FUNCTION_BLOCK FB_working
VAR_INPUT
	lightcurtain_mute_left	: BOOL;
	lightcurtain_mute_right	: BOOL;
	pre_tote_status			: ToteStatus;//roller -1 totestatus=ready
	next_tote_status		: ToteStatus;//roller +1 totestatus=empty
END_VAR
VAR_OUTPUT
	status			: MachineStatus := MachineStatus.STOPPED;
	workflow_status	: ToteSubsystemWorkflowStatus := ToteSubsystemWorkflowStatus.UNKNOWN;
	error_status	: OrderToteErrorStatus := OrderToteErrorStatus.UNKNOWN;	
	tote_status		: ToteStatus;
END_VAR
VAR
	current_tote_status	: ToteStatus;
	ton_timeout			: TON;	
	eStates				: E_WorkingStates	:= E_WorkingStates.IDLE;
	eStateTemp			: E_WorkingStates	:= E_WorkingStates.IDLE;
	iStateTemp			: INT;
	sStateTemp			: STRING;
	errorMessage		: STRING;
	xError				: BOOL;
	iMethod_test		: INT;

	xLoading			: BOOL;
	xUnloading			: BOOL;
///////

	valve_lift			: Valve;
	roller_inbound		: Inbound;
	roller_outbound		: Outbound;
	roller_outbound_end	: Outbound;
	sensor_openbag_detection	: ARRAY[0..7] OF BOOL;
	sensor_cover				: ARRAY[0..1] OF BOOL;
	EDM_KA10			: BOOL;
	mcAxis_lift 		: FB_MotionAxis_MC;
	st_mcAxis_lift 		: ST_MotionAxis_MC;
	AxisRef_lift		: AXIS_REF;
	mcAxis_bag 			: FB_MotionAxis_MC;
	st_mcAxis_bag		: ST_MotionAxis_MC;
	AxisRef_bag			: AXIS_REF;	
	event				: ST_EVENT;
	rt_error			: R_TRIG;
	eTransfer			: E_Transfer;
	
	
	bStopped				: BOOL;
END_VAR
VAR CONSTANT
	rPos_lift_up			: REAL	:= 120;
	rPos_lift_down			: REAL	:= 0;
	rPos_bag_opened			: REAL	:= 45;
	rPos_bag_closed			: REAL	:= 0;
	sComponent_name			: STRING := 'fb_working';
END_VAR

M_mapping();

rt_error(CLK:=(roller_inbound.roller.err OR roller_outbound.roller.err OR roller_outbound_end.roller.err OR st_mcAxis_lift.mcReadStatus.Error 
				OR st_mcAxis_bag.mcReadStatus.Error) AND MAIN.eState<>E_SystemManager.RESET_SAFETY);//roller will trig error while power on
IF rt_error.Q THEN
	xError	:= TRUE;
	eStates	:= E_WorkingStates.ERROR;
END_IF

IF NOT(roller_inbound.photo_sensor_mute.Q OR roller_inbound.photo_sensor.Q OR roller_outbound.photo_sensor.Q) THEN
	current_tote_status	:= ToteStatus.EMPTY;
END_IF
IF NOT roller_inbound.photo_sensor_mute.Q AND roller_inbound.photo_sensor.Q AND NOT roller_outbound.photo_sensor.Q THEN
	current_tote_status	:= ToteStatus.READY;
END_IF



IF eStates=E_WorkingStates.IDLE THEN
	bStopped	:= TRUE;
ELSE
	bStopped	:= FALSE;
END_IF
CASE iMethod_test OF
	0:
	;
	1:		
		IF 	M_load() THEN
			iMethod_test	:= 0;
		END_IF
	2:
		IF 	M_bag_open() THEN
			iMethod_test	:= 0;
		END_IF
	3:
		IF 	M_unload() THEN
			iMethod_test	:= 0;
		END_IF
		
END_CASE

METHOD M_agingTest : BOOL
VAR_INPUT
	
END_VAR
M_AgingTest	:= FALSE;
//////////////////////////////////////////////////////////timeout//////////////////////////////////////////
iStateTemp	:= eStateTemp;
ton_timeout();
IF eStates<>E_WorkingStates.IDLE AND eStates<>E_WorkingStates.ERROR THEN
	IF eStateTemp=eStates THEN
		ton_timeout.IN	:=TRUE;
	ELSE
		ton_timeout.IN	:=FALSE;
		eStateTemp	:= eStates;
	END_IF
ELSE
	ton_timeout.IN	:=FALSE;
END_IF
IF ton_timeout.Q THEN	
	ton_timeout.IN	:=FALSE;
	CASE eStates OF
		E_WorkingStates.AGING_STATE_0:		
			errorMessage	:= CONCAT('wait loading timeout.->fb_loading ',INT_TO_STRING(iStateTemp));
		E_WorkingStates.AGING_STATE_1:		
			errorMessage	:= CONCAT('wait unloading timeout.->fb_loading ',INT_TO_STRING(iStateTemp));
	END_CASE
	IF eStates<>E_WorkingStates.WAIT AND eStates<>E_WorkingStates.WAIT_1 THEN
		//eStates	:= E_WorkingStates.ERROR;
		;
	END_IF
END_IF
CASE eStates OF
	E_WorkingStates.IDLE:
		eStates	:= E_WorkingStates.AGING_STATE_0;
	E_WorkingStates.AGING_STATE_0:
		ton_timeout.PT	:= T#2S;
		st_mcAxis_bag.mcMoveAbsolute.Execute	:= TRUE;						
		st_mcAxis_bag.rActualPosSet	:= rPos_bag_closed;
		st_mcAxis_bag.rVelocitySet	:= 100;
		st_mcAxis_lift.mcMoveAbsolute.Execute	:= TRUE;	
		st_mcAxis_lift.rActualPosSet	:= rPos_lift_up;
		st_mcAxis_lift.rVelocitySet	:= 100;	
		roller_inbound.roller.forward			:= TRUE;
		roller_inbound.roller.backward			:= FALSE;
		roller_outbound.roller.forward			:= TRUE;
		roller_outbound_end.roller.forward		:= TRUE;
		roller_outbound_end.roller.backward		:= FALSE;			
		IF st_mcAxis_bag.mcMoveAbsolute.Done AND st_mcAxis_lift.mcMoveAbsolute.Done AND ton_timeout.Q THEN
			eStates	:= E_WorkingStates.WAIT;
		END_IF			
	E_WorkingStates.WAIT:
		roller_inbound.roller.forward			:= FALSE;
		roller_inbound.roller.backward			:= FALSE;
		roller_outbound.roller.forward			:= FALSE;
		roller_outbound.roller.backward			:= FALSE;
		roller_outbound_end.roller.forward		:= FALSE;
		roller_outbound_end.roller.backward		:= FALSE;	
		st_mcAxis_bag.mcMoveAbsolute.Execute	:= FALSE;
		st_mcAxis_lift.mcMoveAbsolute.Execute	:= FALSE;		
		ton_timeout.PT	:= T#1S;
		IF ton_timeout.Q THEN
			eStates	:= E_WorkingStates.AGING_STATE_1;
		END_IF
	E_WorkingStates.AGING_STATE_1:
		ton_timeout.PT	:= T#2S;
		st_mcAxis_bag.mcMoveAbsolute.Execute	:= TRUE;						
		st_mcAxis_bag.rActualPosSet	:= rPos_bag_opened;
		st_mcAxis_bag.rVelocitySet	:= 100;
		st_mcAxis_lift.mcMoveAbsolute.Execute	:= TRUE;
		st_mcAxis_lift.rActualPosSet	:= rPos_lift_down;
		st_mcAxis_lift.rVelocitySet	:= 100;	
		roller_inbound.roller.forward			:= TRUE;
		roller_inbound.roller.backward			:= TRUE;
		roller_outbound.roller.backward			:= TRUE;
		roller_outbound_end.roller.forward		:= TRUE;
		roller_outbound_end.roller.backward		:= TRUE;			
		IF st_mcAxis_bag.mcMoveAbsolute.Done AND st_mcAxis_lift.mcMoveAbsolute.Done AND ton_timeout.Q THEN
			eStates	:= E_WorkingStates.WAIT_1;
		END_IF	
	E_WorkingStates.WAIT_1:
		ton_timeout.PT	:= T#1S;
		roller_inbound.roller.forward			:= FALSE;
		roller_inbound.roller.backward			:= FALSE;
		roller_outbound.roller.forward			:= FALSE;
		roller_outbound.roller.backward			:= FALSE;
		roller_outbound_end.roller.forward		:= FALSE;
		roller_outbound_end.roller.backward		:= FALSE;	
		st_mcAxis_bag.mcMoveAbsolute.Execute	:= FALSE;
		st_mcAxis_lift.mcMoveAbsolute.Execute	:= FALSE;		
		IF ton_timeout.Q THEN
			eStates	:= E_WorkingStates.IDLE;
		END_IF		
	E_WorkingStates.DONE:
		;
	E_WorkingStates.ERROR:
		;
	
END_CASE
END_METHOD

METHOD M_bag_close : BOOL
VAR_INPUT
END_VAR
END_METHOD

METHOD M_bag_open : BOOL
VAR_INPUT
END_VAR
M_bag_open	:= FALSE;
ADSLOGSTR(msgCtrlMask:= ADSLOG_MSGTYPE_LOG,msgFmtStr:='bag open',strArg:='MSG ARG');
M_bag_open	:= TRUE;
END_METHOD

METHOD M_checkCondition : BOOL
VAR_INPUT
	condition	: E_Condition;
END_VAR
M_checkCondition	:= FALSE;
CASE condition OF
	E_Condition.NO_TOTE:
	 	IF NOT roller_inbound.photo_sensor.Q THEN
			M_checkCondition	:= TRUE;
		END_IF
	E_Condition.TOTE_IN:
	 	IF roller_inbound.photo_sensor.Q THEN
			M_checkCondition	:= TRUE;
		END_IF		
	E_Condition.READY_LOADING_TOTE:
		IF pre_tote_status=ToteStatus.READY THEN
			M_checkCondition	:= TRUE;
		END_IF
	E_Condition.TOTE_READY:
		IF ABS(st_mcAxis_lift.mcReadActualPosition.Position-rPos_lift_down)<1 AND ABS(st_mcAxis_bag.mcReadActualPosition.Position-rPos_bag_opened)<1 
			AND roller_inbound.photo_sensor.Q AND NOT roller_inbound.photo_sensor_mute.Q AND NOT roller_outbound.photo_sensor.Q AND valve_lift.retracted THEN
			tote_status	:= ToteStatus.READY;
		ELSE
			IF tote_status = ToteStatus.READY THEN
				tote_status	:= ToteStatus.LOADED;
			END_IF
		END_IF
		IF ABS(st_mcAxis_lift.mcReadActualPosition.Position-rPos_lift_up)<1 AND ABS(st_mcAxis_bag.mcReadActualPosition.Position-rPos_bag_closed)<1 
			AND NOT roller_inbound.photo_sensor.Q AND NOT roller_inbound.photo_sensor_mute.Q AND NOT roller_outbound.photo_sensor.Q AND valve_lift.retracted THEN
			tote_status	:= ToteStatus.EMPTY;	
		END_IF	
		M_checkCondition	:= TRUE;
END_CASE
END_METHOD

METHOD M_init : BOOL
VAR_INPUT
END_VAR
M_init	:= FALSE;
event.sMethod	:= 'init';
xError	:= FALSE;
st_mcAxis_bag.mcStop.Execute	:= FALSE;
st_mcAxis_bag.mcReset.Execute	:= TRUE;
st_mcAxis_lift.mcStop.Execute	:= FALSE;
st_mcAxis_lift.mcReset.Execute	:= TRUE;
error_status	:= OrderToteErrorStatus.NO_ERROR;

eStates	:= E_WorkingStates.IDLE;
M_init	:= TRUE;
END_METHOD

METHOD M_load : BOOL
VAR_INPUT
END_VAR
VAR_OUTPUT 

END_VAR
M_load := FALSE;
event.sMethod	:= 'load';
//////////////////////////////////////////////////////////timeout//////////////////////////////////////////
iStateTemp	:= eStateTemp;
sStateTemp	:= INT_TO_STRING(iStateTemp);
ton_timeout();
IF eStates<>E_WorkingStates.IDLE AND eStates<>E_WorkingStates.ERROR THEN
	IF eStateTemp=eStates THEN
		ton_timeout.IN	:=TRUE;
	ELSE
		ton_timeout.IN	:=FALSE;
		IF GVL.bAck_stop THEN
			roller_inbound.roller.forward	:= FALSE;
			RETURN;			
		END_IF
		eStateTemp	:= eStates;	
	END_IF
ELSE
	ton_timeout.IN	:=FALSE;
END_IF
IF ton_timeout.Q THEN	
	ton_timeout.IN	:=FALSE;
	CASE eStates OF		
		E_WorkingStates.BAG_OPEN_UP:	
			event.sEventType	:= 'error';
			event.sEvent_MSG	:= CONCAT('BAG_OPEN_UP ','timeout');
			event.sStepID		:= sStateTemp;
		E_WorkingStates.BAG_CLOSE:	
			event.sEventType	:= 'error';
			event.sEvent_MSG	:= CONCAT('BAG_CLOSE ','timeout');
			event.sStepID		:= sStateTemp;					
		E_WorkingStates.TOTE_LIFT_DOWN:			
			event.sEventType	:= 'error';
			event.sEvent_MSG	:= CONCAT('TOTE_LIFT_DOWN ','timeout');
			event.sStepID		:= sStateTemp;
		E_WorkingStates.WAIT_NEW_TOTE://wait empty and trig signal
			;
		E_WorkingStates.TOTE_LOAD:	
			event.sEventType	:= 'error';
			event.sEvent_MSG	:= CONCAT('TOTE_LOAD ','timeout');
			event.sStepID		:= sStateTemp;
		E_WorkingStates.WAIT:
			;
		E_WorkingStates.BAG_OPEN_DOWN:
			event.sEventType	:= 'error';
			event.sEvent_MSG	:= CONCAT('BAG_OPEN_DOWN ','timeout');
			event.sStepID		:= sStateTemp;			
		E_WorkingStates.BAG_OPEN:			
			event.sEventType	:= 'error';
			event.sEvent_MSG	:= CONCAT('BAG_OPEN ','timeout');
			event.sStepID		:= sStateTemp;
		ELSE
			event.sEventType	:= 'error';
			event.sEvent_MSG	:= CONCAT('unknow estate ','timeout');
			event.sStepID		:= sStateTemp;			
	END_CASE
	IF eStates<>E_WorkingStates.WAIT_NEW_TOTE AND eStates<>E_WorkingStates.WAIT THEN
		eStates	:= E_WorkingStates.ERROR;
		error_status	:= OrderToteErrorStatus.MECHANICAL_ERROR;
		Event_add(event);
	END_IF
	
END_IF

CASE eStates OF 
		E_WorkingStates.IDLE:
			ton_timeout.PT	:= T#10S;
			xLoading	:= FALSE;
			xUnloading	:= FALSE;
			st_mcAxis_bag.mcPower.Enable	:= TRUE;
			st_mcAxis_lift.mcPower.Enable	:= TRUE;
			IF st_mcAxis_bag.mcReadStatus.StandStill AND st_mcAxis_lift.mcReadStatus.StandStill THEN
				eStates	:= E_WorkingStates.INIT;
			END_IF			
		E_WorkingStates.INIT:
			xLoading	:= TRUE;		
			st_mcAxis_bag.mcMoveAbsolute.Execute	:= FALSE;
			st_mcAxis_lift.mcMoveAbsolute.Execute	:= FALSE;
			eStates	:= E_WorkingStates.BAG_OPEN_UP;
		E_WorkingStates.BAG_OPEN_UP:	
			st_mcAxis_lift.mcMoveAbsolute.Execute	:= TRUE;		
			st_mcAxis_lift.rActualPosSet	:= rPos_lift_up;
			st_mcAxis_lift.rVelocitySet	:= 250;
			IF st_mcAxis_lift.mcMoveAbsolute.Done THEN
				st_mcAxis_lift.mcMoveAbsolute.Execute	:= FALSE;
				eStates	:= E_WorkingStates.BAG_CLOSE;
			END_IF	
		E_WorkingStates.BAG_CLOSE:	
			st_mcAxis_bag.mcMoveAbsolute.Execute	:= TRUE;		
			st_mcAxis_bag.rActualPosSet	:= rPos_bag_closed;
			st_mcAxis_bag.rVelocitySet	:= 250;
			IF st_mcAxis_bag.mcMoveAbsolute.Done THEN
				st_mcAxis_bag.mcMoveAbsolute.Execute	:= FALSE;
				eStates	:= E_WorkingStates.TOTE_LIFT_DOWN;
			END_IF					
		E_WorkingStates.TOTE_LIFT_DOWN:			
			valve_lift.extend	:= FALSE;
			valve_lift.retract	:= TRUE;
			IF NOT valve_lift.extended AND valve_lift.retracted THEN
				eStates	:= E_WorkingStates.WAIT_NEW_TOTE;
			END_IF	
		E_WorkingStates.WAIT_NEW_TOTE://wait empty and trig signal
			workflow_status	:= ToteSubsystemWorkflowStatus.WAITING_FOR_NEW_TOTE;
			IF NOT(roller_inbound.photo_sensor_mute.Q OR roller_inbound.photo_sensor.Q OR roller_outbound.photo_sensor.Q) THEN
				tote_status	:= ToteStatus.EMPTY;
			END_IF
			IF M_waitCondition(condition:=E_Condition.READY_LOADING_TOTE) THEN
				eStates	:= E_WorkingStates.TOTE_LOAD;
			END_IF
		E_WorkingStates.TOTE_LOAD:	
			workflow_status	:= ToteSubsystemWorkflowStatus.INBOUNDING;
			ton_timeout.PT	:= T#10S;	
			roller_inbound.roller.forward	:= TRUE;
			IF roller_inbound.photo_sensor.Q THEN	
				eStates	:= E_WorkingStates.WAIT;
			END_IF
		E_WorkingStates.WAIT:
			ton_timeout.PT	:= T#300MS;
			roller_inbound.roller.forward	:= TRUE;
			IF ton_timeout.Q THEN
				tote_status	:= ToteStatus.LOADED;
				roller_inbound.roller.forward	:= FALSE;
				eStates	:= E_WorkingStates.BAG_OPEN_DOWN;
			END_IF
		E_WorkingStates.BAG_OPEN_DOWN:
			ton_timeout.PT	:= T#10S;
			workflow_status	:= ToteSubsystemWorkflowStatus.BAG_OPENING;
			st_mcAxis_lift.mcMoveAbsolute.Execute	:= TRUE;		
			st_mcAxis_lift.rActualPosSet	:= rPos_lift_down;
			st_mcAxis_lift.rVelocitySet	:= 250;
			IF st_mcAxis_lift.mcMoveAbsolute.Done THEN
				st_mcAxis_bag.mcMoveAbsolute.Execute	:= FALSE;
				eStates	:= E_WorkingStates.BAG_OPEN;
			END_IF			
		E_WorkingStates.BAG_OPEN:			
			st_mcAxis_bag.mcMoveAbsolute.Execute	:= TRUE;		
			st_mcAxis_bag.rActualPosSet	:= rPos_bag_opened;
			st_mcAxis_bag.rVelocitySet	:= 250;
			IF st_mcAxis_bag.mcMoveAbsolute.Done THEN
				st_mcAxis_bag.mcMoveAbsolute.Execute	:= FALSE;
				eStates	:= E_WorkingStates.DONE;
			END_IF
		E_WorkingStates.DONE:
			tote_status	:= ToteStatus.READY;
			workflow_status	:= ToteSubsystemWorkflowStatus.IDLE;	
			M_load	:= TRUE;
			xLoading	:= FALSE;
			eStates	:= E_WorkingStates.IDLE;
		E_WorkingStates.ERROR:
			xError	:=	TRUE;
			workflow_status	:= ToteSubsystemWorkflowStatus.IDLE;
			roller_inbound.roller.forward		:= FALSE;	
			st_mcAxis_bag.mcMoveAbsolute.Execute	:= FALSE;
			st_mcAxis_lift.mcMoveAbsolute.Execute	:= FALSE;			
			M_load 		:= TRUE;
		
END_CASE
END_METHOD

METHOD M_mapping : BOOL
VAR_INPUT
END_VAR
event.sTime	:= MAIN.Temp_str;
event.sComponent_name	:= sComponent_name;
/////////////////////////////////////digital input////////////////////////////////////////
valve_lift.extended					:= G_IO.arDI[5].Ch[0] OR G_IO.arDI[5].Ch[2];
valve_lift.retracted				:= G_IO.arDI[5].Ch[1] OR G_IO.arDI[5].Ch[3];
roller_inbound.photo_sensor_mute(D:= G_IO.arDI[5].Ch[4],on_ms:=10,off_ms:=100);
roller_inbound.roller.err			:= G_IO.arDI[5].Ch[5];
roller_inbound.photo_sensor(D:= G_IO.arDI[5].Ch[6],on_ms:=100,off_ms:=100);
roller_outbound.roller.err			:= G_IO.arDI[5].Ch[7];
roller_outbound.photo_sensor(D:= G_IO.arDI[5].Ch[8],on_ms:=100,off_ms:=500);		
sensor_openbag_detection[0]			:= G_IO.arDI[5].Ch[9];
sensor_openbag_detection[1]			:= G_IO.arDI[5].Ch[10];
sensor_openbag_detection[2]			:= G_IO.arDI[5].Ch[11];
sensor_openbag_detection[3]			:= G_IO.arDI[5].Ch[12];
sensor_openbag_detection[4]			:= G_IO.arDI[5].Ch[13];
sensor_openbag_detection[5]			:= G_IO.arDI[5].Ch[14];
sensor_openbag_detection[6]			:= G_IO.arDI[5].Ch[15];
sensor_openbag_detection[7]			:= G_IO.arDI[6].Ch[0];
sensor_cover[0]						:= G_IO.arDI[6].Ch[1];
sensor_cover[1]						:= G_IO.arDI[6].Ch[2];
EDM_KA10							:= G_IO.arDI[6].Ch[3];
roller_outbound_end.roller.err		:= G_IO.arDI[6].Ch[4];


/////////////////////////////////////digital output////////////////////////////////////////
G_IO.arDO[5].Ch[0]	:= valve_lift.extend;
G_IO.arDO[5].Ch[1]	:= valve_lift.retract;
G_IO.arDO[5].Ch[2]	:= roller_inbound.roller.forward;
G_IO.arDO[5].Ch[3]	:= roller_inbound.roller.backward;
G_IO.arDO[5].Ch[4]	:= roller_outbound.roller.forward;
G_IO.arDO[5].Ch[5]	:= roller_outbound.roller.backward;
G_IO.arDO[5].Ch[6]	:= roller_outbound_end.roller.forward;
G_IO.arDO[5].Ch[7]	:= roller_outbound_end.roller.backward;
G_IO.arDO[5].Ch[8]	:= lightcurtain_mute_left;
G_IO.arDO[5].Ch[9]	:= lightcurtain_mute_right;



/////////////////////////////////////axis config////////////////////////////////////////
mcAxis_lift
(
	ZSN		:=  TRUE OR st_mcAxis_lift.xHoming, //TODO link to digital input
	ZSP		:=  TRUE OR st_mcAxis_lift.xHoming, //TODO link to digital input
	IN_OUT	:= st_mcAxis_lift	, 
	AXIS	:= AxisRef_lift	, 
);
st_mcAxis_lift.bPosSensorShow	:= TRUE;
st_mcAxis_lift.bNegSensorShow	:= TRUE;
st_mcAxis_lift.rMaxAcceleration	:= 50000;
st_mcAxis_lift.rMaxDeceleration	:= 50000;
st_mcAxis_lift.rMaxJerk			:= 500000;
st_mcAxis_lift.rAcceleration	:= 2500;
st_mcAxis_lift.rDeceleration	:= 2500;
st_mcAxis_lift.rJerk			:= 12500;
st_mcAxis_lift.rMaxVelocity		:= 100;
st_mcAxis_lift.rMaxDistance		:= 50;
st_mcAxis_lift.bPosSen	:= TRUE ;//TODO link to digital input
st_mcAxis_lift.bNegSen	:= TRUE ;//TODO link to digital input
st_mcAxis_lift.mcHome.bCalibrationCam	:= TRUE;//TODO link to digital input origin
st_mcAxis_lift.bPositionSensor	:= TRUE;//TODO link to digital input origin
st_mcAxis_lift.bdirFW	:= TRUE;
st_mcAxis_lift.sNetID := '192.168.11.159.5.1';
st_mcAxis_lift.nSlaveAddr	:= 1026;


mcAxis_bag
(
	ZSN		:=  TRUE OR st_mcAxis_bag.xHoming, //TODO link to digital input
	ZSP		:=  TRUE OR st_mcAxis_bag.xHoming, //TODO link to digital input
	IN_OUT	:= st_mcAxis_bag	, 
	AXIS	:= AxisRef_bag	, 
);
st_mcAxis_bag.bPosSensorShow	:= TRUE;
st_mcAxis_bag.bNegSensorShow	:= TRUE;
st_mcAxis_bag.rMaxAcceleration	:= 50000;
st_mcAxis_bag.rMaxDeceleration	:= 50000;
st_mcAxis_bag.rMaxJerk			:= 500000;
st_mcAxis_bag.rAcceleration	:= 2500;
st_mcAxis_bag.rDeceleration	:= 2500;
st_mcAxis_bag.rJerk			:= 12500;
st_mcAxis_bag.rMaxVelocity		:= 100;
st_mcAxis_bag.rMaxDistance		:= 50;
st_mcAxis_bag.bPosSen	:= TRUE ;//TODO link to digital input
st_mcAxis_bag.bNegSen	:= TRUE ;//TODO link to digital input
st_mcAxis_bag.mcHome.bCalibrationCam	:= TRUE;//TODO link to digital input origin
st_mcAxis_bag.bPositionSensor	:= TRUE;//TODO link to digital input origin
st_mcAxis_bag.bdirFW	:= TRUE;
st_mcAxis_bag.sNetID := '192.168.11.159.5.1';
st_mcAxis_bag.nSlaveAddr	:= 1027;

IF MAIN.firstCycle THEN
	st_mcAxis_bag.mcPower.Enable	:= TRUE;
	st_mcAxis_lift.mcPower.Enable	:= TRUE;	
END_IF
END_METHOD

METHOD M_reset : BOOL
VAR_INPUT
END_VAR
M_reset	:= FALSE;
ton_timeout.IN	:= FALSE;
event.sMethod	:= 'reset';
error_status	:= OrderToteErrorStatus.NO_ERROR;
IF xError THEN
	st_mcAxis_bag.mcStop.Execute	:= FALSE;
	st_mcAxis_bag.mcReset.Execute	:= TRUE;
	st_mcAxis_lift.mcStop.Execute	:= FALSE;
	st_mcAxis_lift.mcReset.Execute	:= TRUE;
	IF eStates<>E_WorkingStates.IDLE THEN
		eStates	:= eStateTemp;//continue
	END_IF
		
	xError	:= FALSE;
ELSE
	;
END_IF

//todo:check if reset successful
M_reset	:= TRUE;
END_METHOD

METHOD M_run : BOOL
VAR_INPUT
END_VAR
//
IF M_checkCondition(condition:= E_Condition.NO_TOTE) THEN
	;
END_IF
//check no tote of working
//wait new tote of loading
//tote load
END_METHOD

METHOD M_runStart : BOOL
VAR_INPUT
END_VAR
M_runStart	:= FALSE;
st_mcAxis_bag.mcPower.Enable	:= TRUE;
st_mcAxis_lift.mcPower.Enable	:= TRUE;

current_tote_status	:= ToteStatus.UNKNOWN;
M_checkCondition(condition:=E_Condition.TOTE_READY);


IF st_mcAxis_bag.mcReadStatus.StandStill AND st_mcAxis_lift.mcReadStatus.StandStill THEN
	M_runStart	:= TRUE;
END_IF
M_runStart	:= TRUE;
END_METHOD

METHOD M_safetyEvent : BOOL
VAR_INPUT
END_VAR
M_safetyEvent	:= FALSE;

roller_inbound.roller.forward			:= FALSE;
roller_inbound.roller.backward			:= FALSE;
roller_outbound.roller.forward			:= FALSE;
roller_outbound.roller.backward			:= FALSE;
roller_outbound_end.roller.forward		:= FALSE;	
roller_outbound_end.roller.backward		:= FALSE;	
st_mcAxis_bag.mcMoveAbsolute.Execute	:= FALSE;
st_mcAxis_lift.mcMoveAbsolute.Execute	:= FALSE;	
st_mcAxis_bag.mcStop.Execute	:= TRUE;
st_mcAxis_lift.mcStop.Execute	:= TRUE;

M_safetyEvent	:= TRUE;
END_METHOD

METHOD M_toteLoad : BOOL
VAR_INPUT
END_VAR
M_toteLoad	:= FALSE;
IF roller_inbound.photo_sensor.Q THEN
	roller_inbound.roller.forward	:= FALSE;
	ADSLOGSTR(msgCtrlMask:= ADSLOG_MSGTYPE_LOG,msgFmtStr:='tote load finish',strArg:='MSG ARG');
ELSE
	roller_inbound.roller.forward	:= TRUE;
	ADSLOGSTR(msgCtrlMask:= ADSLOG_MSGTYPE_LOG,msgFmtStr:='tote load start',strArg:='MSG ARG');
	M_toteLoad	:= TRUE;
END_IF
END_METHOD

METHOD M_toteUnload : BOOL
VAR_INPUT
END_VAR
M_toteUnload	:= FALSE;

CASE eStates OF 
		E_WorkingStates.TOTE_LIFT_UP:
			valve_lift.extend	:= TRUE;
			valve_lift.retract	:= FALSE;
			IF valve_lift.extended AND NOT valve_lift.retracted THEN
				eStates	:= E_WorkingStates.TOTE_UNLOAD;
			END_IF
		E_WorkingStates.TOTE_OUT:
			IF roller_outbound.photo_sensor.Q THEN
				roller_outbound.roller.forward	:= FALSE;
				M_toteUnload	:= TRUE;
			ELSE
				roller_outbound.roller.forward	:= TRUE;
			END_IF	
		E_WorkingStates.TOTE_LIFT_DOWN:	
			valve_lift.extend	:= FALSE;
			valve_lift.retract	:= TRUE;
			IF NOT valve_lift.extended AND valve_lift.retracted THEN
				M_toteUnload	:= TRUE;
			END_IF	
END_CASE
END_METHOD

METHOD M_unload : BOOL
VAR_INPUT
END_VAR
VAR_OUTPUT 

END_VAR
//initialize
//bag_open lift up & bag_open_home
//tote lift up
//outbound
//tote lift down
//done
M_unload := FALSE;
event.sMethod	:= 'unload';
//////////////////////////////////////////////////////////timeout//////////////////////////////////////////
iStateTemp	:= eStateTemp;
sStateTemp	:= INT_TO_STRING(iStateTemp);
ton_timeout();
IF eStates<>E_WorkingStates.IDLE AND eStates<>E_WorkingStates.ERROR  THEN
	IF eStateTemp=eStates THEN
		ton_timeout.IN	:=TRUE;
	ELSE
		ton_timeout.IN	:=FALSE;
		IF GVL.bAck_stop THEN
			roller_outbound.roller.forward	:= FALSE;
			roller_outbound_end.roller.forward	:= FALSE;
			RETURN;		
		END_IF
		eStateTemp	:= eStates;
	END_IF
ELSE
	ton_timeout.IN	:=FALSE;
END_IF
IF ton_timeout.Q THEN	
	ton_timeout.IN	:=FALSE;
	CASE eStates OF
	
		E_WorkingStates.WAIT_UNLOADING://wait signal from logtech and app to unload the tote
			;
		E_WorkingStates.BAG_OPEN_UP:	
			event.sEventType	:= 'error';
			event.sEvent_MSG	:= CONCAT('BAG_OPEN_UP ','timeout');
			event.sStepID		:= sStateTemp;
		E_WorkingStates.BAG_CLOSE:	
			event.sEventType	:= 'error';
			event.sEvent_MSG	:= CONCAT('BAG_CLOSE or TOTE_LIFT_UP ','timeout');
			event.sStepID		:= sStateTemp;						
		E_WorkingStates.TOTE_LIFT_UP:
			event.sEventType	:= 'error';
			event.sEvent_MSG	:= CONCAT('TOTE_LIFT_UP ','timeout');
			event.sStepID		:= sStateTemp;
		E_WorkingStates.TOTE_UNLOAD:
			event.sEventType	:= 'error';
			event.sEvent_MSG	:= CONCAT('TOTE_UNLOAD ','timeout');
			event.sStepID		:= sStateTemp;

		E_WorkingStates.WAIT_SENSOR_OFF:	
			event.sEventType	:= 'error';
			event.sEvent_MSG	:= CONCAT('WAIT_SENSOR_OFF ','timeout');
			event.sStepID		:= sStateTemp;	
		E_WorkingStates.TOTE_LIFT_DOWN:
			event.sEventType	:= 'error';
			event.sEvent_MSG	:= CONCAT('TOTE_LIFT_DOWN ','timeout');
			event.sStepID		:= sStateTemp;
		ELSE
			event.sEventType	:= 'error';
			event.sEvent_MSG	:= CONCAT('unknow estate ','timeout');
			event.sStepID		:= sStateTemp;			
	END_CASE
	IF eStates<>E_WorkingStates.IDLE AND eStates<>E_WorkingStates.WAIT_UNLOADING THEN
		eStates	:= E_WorkingStates.ERROR;
		error_status	:= OrderToteErrorStatus.MECHANICAL_ERROR;
		Event_add(event);
	END_IF
	
END_IF

CASE eStates OF 
		E_WorkingStates.IDLE:
			ton_timeout.PT	:= T#10S;
			xLoading	:= FALSE;
			xUnloading	:= FALSE;
			eStates	:= E_WorkingStates.INIT;
		E_WorkingStates.INIT:	
			xUnloading	:= TRUE;
			st_mcAxis_bag.mcMoveAbsolute.Execute	:= FALSE;
			st_mcAxis_lift.mcMoveAbsolute.Execute	:= FALSE;
			eStates	:= E_WorkingStates.WAIT_UNLOADING;
		E_WorkingStates.WAIT_UNLOADING://wait signal from logtech and app to unload the tote
			workflow_status	:= ToteSubsystemWorkflowStatus.WAITING_FOR_UNLOADING;
			tote_status	:= ToteStatus.READY;
			eStates	:= E_WorkingStates.BAG_OPEN_UP;	
		E_WorkingStates.BAG_OPEN_UP:	
			workflow_status	:= ToteSubsystemWorkflowStatus.OUTBOUNDING;	
			tote_status	:= ToteStatus.LOADED;		
			st_mcAxis_lift.mcMoveAbsolute.Execute	:= TRUE;		
			st_mcAxis_lift.rActualPosSet	:= rPos_lift_up;
			st_mcAxis_lift.rVelocitySet	:= 250;
			IF st_mcAxis_lift.mcMoveAbsolute.Done THEN
				eStates	:= E_WorkingStates.BAG_CLOSE;
			END_IF		
		E_WorkingStates.BAG_CLOSE:	
			st_mcAxis_bag.mcMoveAbsolute.Execute	:= TRUE;		
			st_mcAxis_bag.rActualPosSet	:= rPos_bag_closed;
			st_mcAxis_bag.rVelocitySet	:= 250;
			valve_lift.extend	:= TRUE;
			valve_lift.retract	:= FALSE;
			IF st_mcAxis_bag.mcMoveAbsolute.Done AND valve_lift.extended AND NOT valve_lift.retracted THEN
				st_mcAxis_bag.mcMoveAbsolute.Execute	:= FALSE;
				eStates	:= E_WorkingStates.TOTE_UNLOAD;
			END_IF							
//		E_WorkingStates.TOTE_LIFT_UP:
//			ton_timeout.PT	:= T#5S;
//			valve_lift.extend	:= TRUE;
//			valve_lift.retract	:= FALSE;
//			IF valve_lift.extended AND NOT valve_lift.retracted THEN
//				eStates	:= E_WorkingStates.TOTE_UNLOAD;
//			END_IF
		E_WorkingStates.TOTE_UNLOAD:
			ton_timeout.PT	:= T#5S;
			roller_outbound.roller.forward		:= TRUE;
			roller_outbound_end.roller.forward	:= TRUE;
			IF roller_outbound.photo_sensor.Q THEN
				eStates	:= E_WorkingStates.WAIT_SENSOR_OFF;			
			END_IF	
		E_WorkingStates.WAIT_SENSOR_OFF:
			roller_outbound.roller.forward		:= TRUE;
			roller_outbound_end.roller.forward	:= TRUE;	
			IF NOT roller_outbound.photo_sensor.Q THEN
				roller_outbound.roller.forward		:= FALSE;	
				roller_outbound_end.roller.forward	:= FALSE;
				eStates	:= E_WorkingStates.TOTE_LIFT_DOWN;			
			END_IF			
		E_WorkingStates.TOTE_LIFT_DOWN:
			ton_timeout.PT	:= T#5S;	
			valve_lift.extend	:= FALSE;
			valve_lift.retract	:= TRUE;
			IF NOT valve_lift.extended AND valve_lift.retracted THEN
				eStates	:= E_WorkingStates.DONE;
			END_IF				
		E_WorkingStates.DONE:	
			workflow_status	:= ToteSubsystemWorkflowStatus.IDLE;
			tote_status	:= ToteStatus.EMPTY;			
			M_unload	:= TRUE;
			xUnloading	:= FALSE;
			eStates	:= E_WorkingStates.IDLE;
		E_WorkingStates.ERROR:
			xError	:=	TRUE;
			workflow_status	:= ToteSubsystemWorkflowStatus.IDLE;
			roller_outbound.roller.forward		:= FALSE;	
			roller_outbound_end.roller.forward	:= FALSE;
			st_mcAxis_bag.mcMoveAbsolute.Execute	:= FALSE;
			st_mcAxis_lift.mcMoveAbsolute.Execute	:= FALSE;
			M_unload 		:= TRUE;

		
END_CASE
END_METHOD

METHOD M_waitCondition : BOOL
VAR_INPUT
	condition	: E_Condition;
END_VAR
M_waitCondition	:= FALSE;
CASE condition OF
	E_Condition.NO_TOTE:
	 	IF NOT roller_inbound.photo_sensor.Q THEN
			M_waitCondition	:= TRUE;
		END_IF
	E_Condition.TOTE_IN:
	 	IF roller_inbound.photo_sensor.Q THEN
			M_waitCondition	:= TRUE;
		END_IF	
	E_Condition.READY_LOADING_TOTE:
		IF pre_tote_status=ToteStatus.READY AND GVL.fb_loading.eTransfer=E_Transfer.UNLOAD OR tote_status=ToteStatus.LOADED THEN
			M_waitCondition	:= TRUE;
		END_IF	
END_CASE
END_METHOD

END_FUNCTION_BLOCK

(* stored: Version 1.1.0.1, ProductVersion 3.1.4024.12
   POU FB_working: Id {5476bf73-fb6f-4e63-89b1-2ec0afd3a62f}, SpecialFunc None
   Method M_agingTest: Id {c302c8df-88d7-4884-b79e-724a2f679edf}
   Method M_bag_close: Id {66b5f911-16ac-4932-bbc7-7b12fc8051b5}
   Method M_bag_open: Id {6f59acea-9082-4203-a9b2-cefe10215e2d}
   Method M_checkCondition: Id {f334d666-8f81-40fc-b350-e1376c64bbdc}
   Method M_init: Id {9816fa7a-9c52-4ba9-8037-d612c8e8504d}
   Method M_load: Id {3b4981fb-68b3-4b99-90aa-3986e3b47b1a}
   Method M_mapping: Id {47e6ed7c-b89d-46d1-bd0a-f3c311dd6211}
   Method M_reset: Id {79f562bd-508c-433a-9c3f-c76c9e6cd0fa}
   Method M_run: Id {d589d7a8-9e09-4d7c-95b2-7ebc3d85ecae}
   Method M_runStart: Id {7c0f4dcb-6112-4937-805e-6367eecb6122}
   Method M_safetyEvent: Id {0b8a20f6-fb60-4092-9d2d-ef36588456de}
   Method M_toteLoad: Id {15ef71f7-21f3-44c6-b1a1-c7f688409d7c}
   Method M_toteUnload: Id {929d8c87-be93-4a3b-80c4-23b2766f3017}
   Method M_unload: Id {cb0cfbd0-7970-4d6c-a403-8613470fb781}
   Method M_waitCondition: Id {ed247d89-1b4f-4668-b2d3-5596d020db3a} *)
